TYPE ST_PhysicalInputs :
STRUCT
    // Physical operator controls (standard PLC inputs)
    bStartButton                  : BOOL;
    bStopButton                   : BOOL;

    // Reset and validated safety diagnostics received through TwinSAFE aliases
    bResetButton                  : BOOL;
    bTwoHandsSafe                 : BOOL;
    bSafetyOk                     : BOOL;
    bEmergencyStopOk              : BOOL;
    bMainDoorSafe                 : BOOL;
    bLeftFlapSafe                 : BOOL;
    bRightFlapSafe                : BOOL;
    bFlapsSafe                    : BOOL;
    bFsoeOk                       : BOOL;
    bSafetyLogicOk                : BOOL;
    bAirSupplyOk                  : BOOL;

    // Power and auxiliary diagnostics
    bUp24VPowerSupplyOk         	: BOOL;
    bUs24VPowerSupplyOk         	: BOOL;
    bIvekHeaterControllerAlarm  	: BOOL;
    bSiliconeMinimumLevelSensor1 	: BOOL;
    bSiliconeMinimumLevelSensor2 	: BOOL;

    // Door diagnostics returned by TwinSAFE
    bMainDoorClosed               : BOOL;
    bMainDoorLocked               : BOOL;
    bMainDoorDiagnosticOk         : BOOL;
    bMs6FeedbackOk                : BOOL;
    bAirExhausted                 : BOOL;

    // Part detection
    bGearboxAssemblyPartPresent   : BOOL;
    bReservoirPartPresent         : BOOL;
    bRejectChutePartPresent       : BOOL;

    // Index table
    bIndexPositionSensor1         : BOOL;
    bIndexPositionSensor2         : BOOL;
    bIndexPositionSensor3         : BOOL;
    bIndexReady                   : BOOL;
    bIndexLocked                  : BOOL;
    bIndexCompletedSensor         : BOOL;
    bIndexSupportExtended         : BOOL;
    bIndexSupportRetracted        : BOOL;
    eIndexPosition                : E_TablePosition;

    // Transfer nest support / process tooling cylinder
    bTransferNestSupportCylinderExtended        : BOOL;
    bTransferNestSupportCylinderRetracted       : BOOL;

    // Analog raw values. Engineering-unit scaling is intentionally kept
    // outside the terminal mapping until the sensor ranges are confirmed.
    uiMainAirPressureRaw          : UINT;
    uiSiliconePressureRaw         : UINT;
    uiNozzlePressureRaw           : UINT;
    uiVacuumPressureRaw           : UINT;

    // Puck locker is not shown in EPLAN Rev 1.0. These remain available for
    // future hardware revisions and must stay FALSE while the option is absent.
    bPuckSensorUp                 : BOOL;
    bPuckSensorDown               : BOOL;
END_STRUCT
END_TYPE

(* stored: Version 1.1.0.1, ProductVersion 3.1.4026.18
   DUT ST_PhysicalInputs: Id {d4e9038a-638b-4b93-a8ec-1f818bc84700} *)
